Staubli VAL3: selectProg.pgx

program selectProg(string x_sProg)
  local num l_nSize
  local string l_sEvent
  local num i
  local num l_nIndex
  local string l_sProg
  local num l_nKey
  local string l_sEmpty
begin
  // show the proram list
  call use:clear(0,13)
  //
  call use:stringCopy(l_sEmpty,sList)
  nSelected=-1
  //
  // Build the list
  //
  call prog:getSize(l_nSize)
  for i=0 to l_nSize-1
    call prog:get(l_sEvent,i)
    if l_sEvent!=""
      call listAdd(l_sEvent)
      if l_sEvent==x_sProg
        // select the default
        nSelected=i
      endIf
    endIf
  endFor
  //
  // Show the list
  //
  // define your list size for default
  call use:setSizeList(10,0,17,10)
  //
  call use:listcreate("PROG")
  call use:listadd(sList)
  call use:selectNewField(nSelected,0,0)
  //
  call use:type(35,13,"RESET")
  do
    l_nKey=get()
    call use:listevent(l_nKey,l_nIndex,l_sProg)
    if l_nKey==278
      jEditPoint.sProgram=""
      return
    endIf
  until l_nKey==255 or l_nKey==270
  // save the data
  if l_nKey!=255
    jEditPoint.sProgram=l_sProg
  endIf
end
